PROGRAM Work
VAR
	fbHVACWork: FB_HVACWork;
	eDataSecurityType: E_HVACDataSecurityType;
	bSetDefault: BOOL;
	bOn: BOOL;
	bResetHours: BOOL;
	bResetCount: BOOL;
	dtSystemTime: DATE_AND_TIME;
	bStartWarnLevel: BOOL;
	bStartAlarmLevel: BOOL;
	bSysTakt1Hz: BOOL;
	bReset: BOOL;
	rHours: REAL;
	uiCount: UINT;
	uiWarnLevel: UINT;
	uiAlarmLevel: UINT;
	bEnableWarnLevel: BOOL;
	bEnableAlarmLevel: BOOL;
	bQAlarmLevel: BOOL;
	bQWarnLevel: BOOL;
	bInvalidParameter: BOOL;
END_VAR

fbHVACWork(
	eDataSecurityType:=eDataSecurityType, 
	bSetDefault:=bSetDefault, 
	bOn:=bOn, 
	bResetHours:=bResetHours, 
	bResetCount:=bResetCount, 
	dtSystemTime:=dtSystemTime, 
	bStartWarnLevel:=bStartWarnLevel, 
	bStartAlarmLevel:=bStartAlarmLevel, 
	bSysTakt1Hz:=bSysTakt1Hz, 
	bReset:=bReset, 
	rHours:=rHours, 
	uiCount:=uiCount, 
	uiWarnLevel:=uiWarnLevel, 
	uiAlarmLevel:=uiAlarmLevel, 
	bEnableWarnLevel:=bEnableWarnLevel, 
	bEnableAlarmLevel:=bEnableAlarmLevel, 
	bQAlarmLevel=>bQAlarmLevel, 
	bQWarnLevel=>bQWarnLevel, 
	bInvalidParameter=>bInvalidParameter);

END_PROGRAM

(* stored: Version 1.1.0.1, ProductVersion 3.1.4024.3
   POU Work: Id {b9737889-12cb-4d36-b1d4-37b8d941cb2b}, SpecialFunc None *)
